(* IEC 61131-3 sources: AutomationLab/ConveyerObject/Model/Logic, 1 file *)

(* ---- AlwaysOn.st ---- *)
FUNCTION AlwaysOn : BOOL
VAR_INPUT
	Allow:BOOL;
END_VAR
VAR
END_VAR

AlwaysOn := Allow;
